{attribute 'OPC.UA.DA.StructuredType':=1}
TYPE ST_GripperSpecific :
STRUCT
    TargetPosition  : REAL := 0.0;
    ActualPosition  : REAL := 0.0;

    TargetForce     : REAL := 0.0;
    ActualForce     : REAL := 0.0;

    ObjectDetected  : BOOL := FALSE;
END_STRUCT
END_TYPE

(* stored: Version 1.1.0.1, ProductVersion 3.1.4026.18
   DUT ST_GripperSpecific: Id {160838c9-eb4f-4005-8e3e-1344d5051a0c} *)
